{attribute 'GeneratedUsingTerminal: EL2521-0124-0016'}
{attribute addProperty BoxType "EL2521-0124-0016"}
{attribute addProperty Id "EtcSlaveTerminalBasePTO_StatusAT %I*PTO_Status_C6D3EC315ENC_Status_compactAT %I*ENC_Status_compact_64F890EB11PLS_StatusAT %I*PLS_Status_A60F49334PTO_ControlAT %Q*PTO_Control_392B4D2E5ENC_Control_compactAT %Q*ENC_Control_compact_DC4E290B5PLS_Control_compactAT %Q*PLS_Control_compact_DC91A7B86WcStateAT %I*WcState_9091E0EB2InfoDataAT %I*InfoData_32EB74EA10"}
{attribute addProperty CRC "485458763"}
{attribute addProperty Size "48"}
TYPE EL2521_1CEF834B EXTENDS EtcSlaveTerminalBase :
STRUCT
	{attribute addProperty Name "PTO_Status"}
	PTO_Status : PTO_Status_C6D3EC31;
	{attribute addProperty Name "ENC_Status_compact"}
	ENC_Status_compact : ENC_Status_compact_64F890EB;
	{attribute addProperty Name "PLS_Status"}
	PLS_Status : PLS_Status_A60F4933;
	{attribute addProperty Name "PTO_Control"}
	PTO_Control : PTO_Control_392B4D2E;
	{attribute addProperty Name "ENC_Control_compact"}
	ENC_Control_compact : ENC_Control_compact_DC4E290B;
	{attribute addProperty Name "PLS_Control_compact"}
	PLS_Control_compact : PLS_Control_compact_DC91A7B8;
	{attribute addProperty Name "WcState"}
	WcState : WcState_9091E0EB;
	{attribute addProperty Name "InfoData"}
	InfoData : InfoData_32EB74EA;
END_STRUCT
END_TYPE

(* stored: Version 1.2.0.0, ProductVersion 3.1.4024.9
   DUT EL2521_1CEF834B: Id {ca4a3a4c-e4e6-4f22-b54d-df73dc55530f} *)
